SUBAPPLICATION Uebung_015 (* Subapplication Type *)
  (* Standard: 61499-2 *)
  (* Version 1.0, 2023-10-23, franz *)
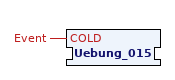
  EVENT_INPUT
    COLD;
  END_EVENT
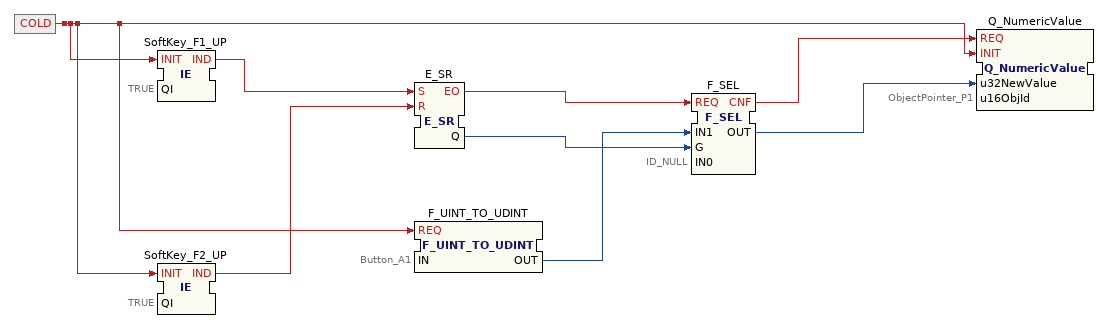
  FBS
    SoftKey_F1_UP : IE(QI := TRUE);
    SoftKey_F2_UP : IE(QI := TRUE);
    E_SR : E_SR;
    F_UINT_TO_UDINT : F_UINT_TO_UDINT(IN := Button_A1);
    F_SEL : F_SEL(IN0 := ID_NULL);
    Q_NumericValue : Q_NumericValue(u16ObjId := ObjectPointer_P1);
  END_FBS
  EVENT_CONNECTIONS
    COLD TO SoftKey_F1_UP.INIT;
    COLD TO SoftKey_F2_UP.INIT;
    SoftKey_F1_UP.IND TO E_SR.S;
    SoftKey_F2_UP.IND TO E_SR.R;
    F_SEL.CNF TO Q_NumericValue.REQ;
    E_SR.EO TO F_SEL.REQ;
    COLD TO Q_NumericValue.INIT;
    COLD TO F_UINT_TO_UDINT.REQ;
  END_CONNECTIONS
  DATA_CONNECTIONS
    F_SEL.OUT TO Q_NumericValue.u32NewValue;
    F_UINT_TO_UDINT.OUT TO F_SEL.IN1;
    E_SR.Q TO F_SEL.G;
  END_CONNECTIONS
END_SUBAPPLICATION
